(* IEC 61131-3 sources: AXOpen/src/abstractions/ctrl/src, 3 files *)

(* ---- IAxoLogger.st ---- *)
USING AXOpen.Core;
USING AXOpen.Core;
NAMESPACE AXOpen.Messaging

    TYPE
        eLogLevel : (Verbose, Debug, Information, Warning, Error, Fatal) := Information;
    END_TYPE

    INTERFACE PUBLIC IAxoLogger
        METHOD Log
            VAR_INPUT
                _message : STRING[254];
                _level : eLogLevel;
                _sender : IAxoObject;
            END_VAR
        END_METHOD
    END_INTERFACE
END_NAMESPACE

(* ---- IsNullContext.st ---- *)
NAMESPACE AXOpen.Core
    FUNCTION IsNullContext : BOOL
        VAR_INPUT
            Context : IAxoContext;
        END_VAR
        IF Context = NULL THEN
            IsNullContext := TRUE;
        ELSIF Context.CreateIdentity() = ULINT#0 THEN
            IsNullContext := TRUE;
        ELSE
            IsNullContext := FALSE;
        END_IF;
    END_FUNCTION
END_NAMESPACE

(* ---- NULLs.st ---- *)
USING AXOpen.Rtc;
NAMESPACE AXOpen.Core
    ///<summary>
    /// Provides an empty context for uninitialized objects.
    ///</summary>
    CLASS PUBLIC _NULL_CONTEXT IMPLEMENTS IAxoContext
        VAR PRIVATE
            NULL_RTC : _NULL_RTC;
        END_VAR

        METHOD PUBLIC CreateIdentity : ULINT CreateIdentity := ULINT#0; END_METHOD
        METHOD PUBLIC OpenCycleCount : ULINT OpenCycleCount := ULINT#0; END_METHOD
        METHOD PUBLIC GetRtc : IAxoRtc GetRtc := NULL_RTC; END_METHOD
        METHOD PUBLIC InjectRtc VAR_INPUT Rtc : IAxoRtc; END_VAR ; END_METHOD
    END_CLASS

    ///<summary>
    /// Provides an empty object for uninitialized objects.
    ///</summary>
    CLASS PUBLIC _NULL_OBJECT IMPLEMENTS IAxoObject
        VAR PRIVATE
            NULL_CONTEXT : _NULL_CONTEXT;
        END_VAR
        METHOD PUBLIC GetIdentity : ULINT
            GetIdentity := ULINT#0;
        END_METHOD
        METHOD PUBLIC GetContext : IAxoContext
            GetContext := NULL_CONTEXT;
        END_METHOD
    END_CLASS

    ///<summary>
    /// Provides an empty RTC object for uninitialized RTC.
    ///</summary>
    CLASS PUBLIC _NULL_RTC IMPLEMENTS IAxoRtc
        VAR PRIVATE
            _null_time : LDATE_AND_TIME := LDATE_AND_TIME#1970-01-01-00:00:00.000;
        END_VAR
        METHOD PUBLIC NowUTC : LDATE_AND_TIME
            NowUTC := _null_time;
        END_METHOD
    END_CLASS
END_NAMESPACE
